// TIA Portal V15.1 export
// export: Created 2026-01-15T16:29:48.8769774Z, ExportSetting WithDefaults, WithReadOnly, DisplayName Totally Integrated Automation Portal, DisplayVersion V15.1 Update 8, DisplayName TIA Portal Openness, DisplayVersion V15.1 Update 8, DisplayName STEP 7 Professional, DisplayVersion V15.1 Update 8, DisplayName WinCC Advanced, DisplayVersion V15.1 Update 8
VAR_GLOBAL   // PLC tag table "Default tag table"
END_VAR
